(* PLC project My_First_Project, Unknown Unnamed 1 *)
(* stored: creationDateTime 2020-02-20T16:42:49, modificationDateTime 2020-03-30T20:15:12 *)

PROGRAM My_First_Program
  VAR
    PB1 AT %QX0.0 : BOOL;
    PB2 AT %QX1.0 : BOOL;
    LAMP AT %QX2.0 : BOOL;
  END_VAR

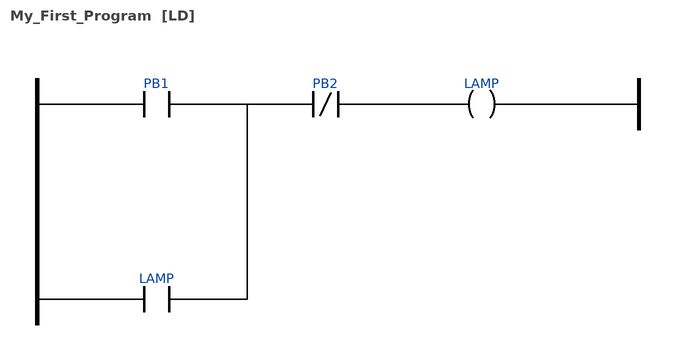
(* LD diagram, written out as Structured Text *)
LAMP := (PB1 OR LAMP) AND NOT PB2;
END_PROGRAM

CONFIGURATION Config0
  RESOURCE Res0 ON PLC
    TASK My_Task(INTERVAL := T#1s, PRIORITY := 0);
    PROGRAM My_Instance WITH My_Task : My_First_Program;
  END_RESOURCE
END_CONFIGURATION
